// SIMATIC S7-200 project (STEP 7-Micro/WIN), CPU 224XP REL 02.01

SYMBOL_TABLE USUARIO1
MARCHA           I0.0
FC1              I0.1
FC2              I0.2
PARO             I0.3
CINTA_1          Q0.0
LED_CINTA_1      Q0.1
CINTA_2          Q0.2
LED_CINTA_2      Q0.3
LED_PARO         Q0.4
END_SYMBOL_TABLE

ORGANIZATION_BLOCK PRINCIPAL:OB1
TITLE=COMENTARIOS DEL PROGRAMA
BEGIN
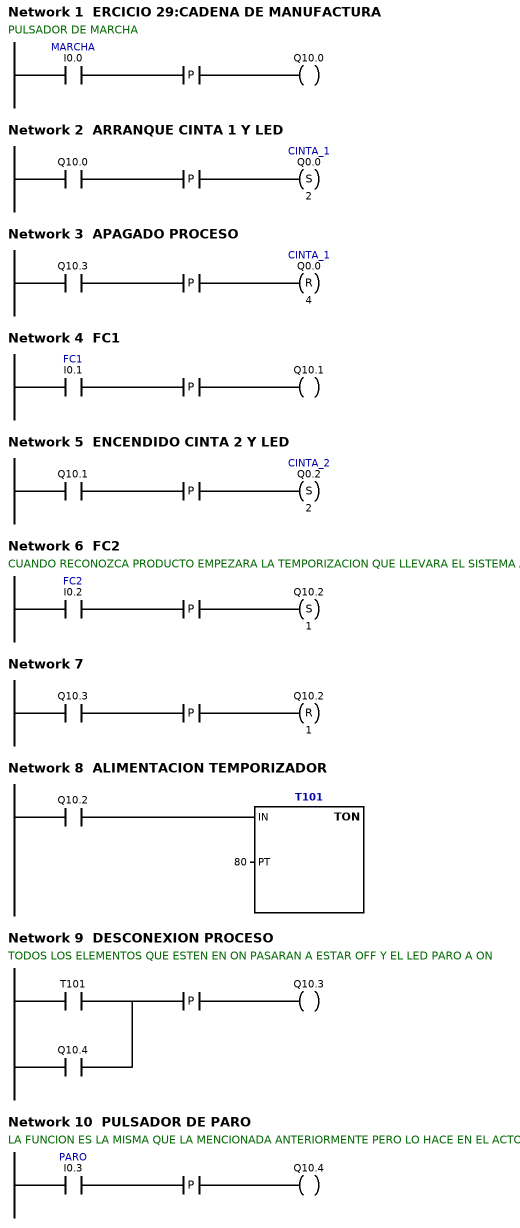
Network 1 // ERCICIO 29:CADENA DE MANUFACTURA
// PULSADOR DE MARCHA
LD     MARCHA:I0.0
EU
=      Q10.0
Network 2 // ARRANQUE CINTA 1 Y LED 
LD     Q10.0
EU
S      CINTA_1:Q0.0, 2
Network 3 // APAGADO PROCESO
LD     Q10.3
EU
R      CINTA_1:Q0.0, 4
Network 4 // FC1
LD     FC1:I0.1
EU
=      Q10.1
Network 5 // ENCENDIDO CINTA 2 Y LED
LD     Q10.1
EU
S      CINTA_2:Q0.2, 2
Network 6 // FC2
// CUANDO RECONOZCA PRODUCTO EMPEZARA LA TEMPORIZACION QUE LLEVARA EL SISTEMA A SITUACION DE REPOSO
LD     FC2:I0.2
EU
S      Q10.2, 1
Network 7
LD     Q10.3
EU
R      Q10.2, 1
Network 8 // ALIMENTACION TEMPORIZADOR
// (network saved uncompiled; LAD cells follow)
// row 0: c0 -| |- Q10.2  c1 --  c2 [TON T101 IN:=power@row0, PT:=80]
// row 1: c2 [box]
Network 9 // DESCONEXION PROCESO
// TODOS LOS ELEMENTOS QUE ESTEN EN ON PASARAN A ESTAR OFF Y EL LED PARO A ON
// (network saved uncompiled; LAD cells follow)
// row 0: c0 -| |- T101 v  c1 -|P|-  c2 -( ) Q10.3
// row 1: c0 -| |- Q10.4 ^
Network 10 // PULSADOR DE PARO 
// LA FUNCION ES LA MISMA QUE LA MENCIONADA ANTERIORMENTE PERO LO HACE EN EL ACTO
LD     PARO:I0.3
EU
=      Q10.4
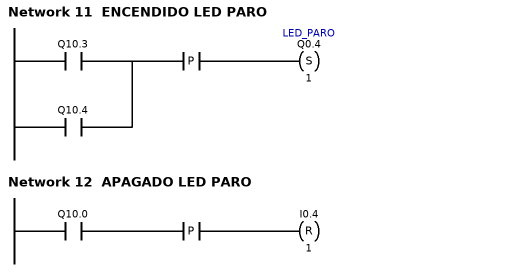
Network 11 // ENCENDIDO LED PARO
LD     Q10.3
O      Q10.4
EU
S      LED_PARO:Q0.4, 1
Network 12 // APAGADO LED PARO
LD     Q10.0
EU
R      I0.4, 1
END_ORGANIZATION_BLOCK
